% RSLogix 500 project DynamicDataExchange.RSS, saved by version 8.30.00.16 %
PROJECT "SIM_PLC"    % processor: Bul.1763 MicroLogix 1100 Series B %

PROGRAM FILES
  LAD 2 "MAIN"  2 rungs
  LAD 3 "CTRL LOGIC"  9 rungs

DATA FILES
  O0 OUTPUT  4 elements
  I1 INPUT  6 elements
  S2 STATUS  66 elements
  B3 BINARY  1 elements
  T4 TIMER  1 elements
  C5 COUNTER  5 elements
  R6 CONTROL  1 elements
  N7 INTEGER  4 elements
  F8 FLOAT  1 elements
  ST9 STRING  8 elements

LADDER 2 "MAIN"
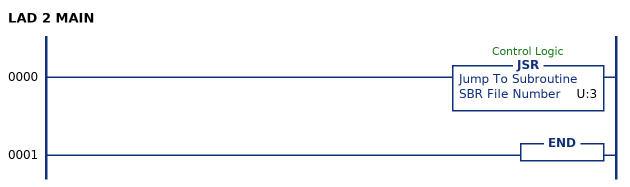
% Rung: 0 %
SOR JSR U:3 EOR
%   U:3  "Control Logic" %
% Rung: 1 %
SOR END EOR

LADDER 3 "CTRL LOGIC"
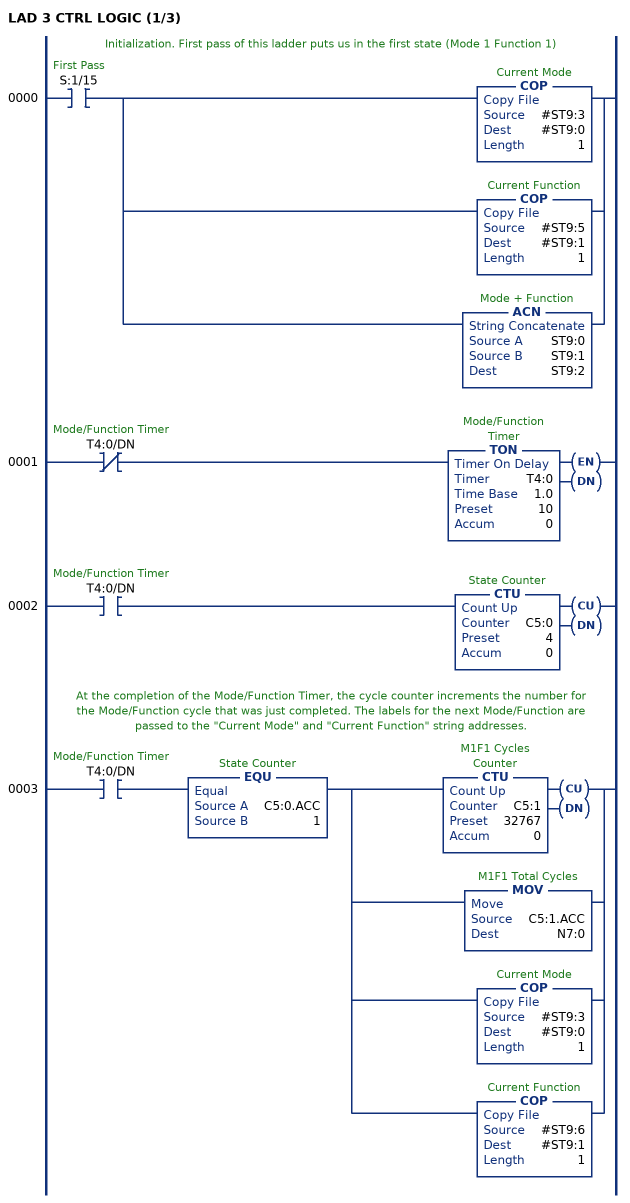
% Rung: 0 %
% Initialization. First pass of this ladder puts us in the first state (Mode 1 Function 1) %
SOR XIC S:1/15 BST COP #ST9:3 #ST9:0 1 NXB COP #ST9:5 #ST9:1 1 NXB ACN ST9:0 ST9:1 ST9:2 BND EOR
%   S:1/15  "First Pass" %
%   ST9:0  "Current Mode" %
%   ST9:1  "Current Function" %
%   ST9:2  "Mode + Function" %
% Rung: 1 %
SOR XIO T4:0/DN TON T4:0 1.0 10 0 EOR
%   T4:0  "Mode/Function Timer" %
% Rung: 2 %
SOR XIC T4:0/DN CTU C5:0 4 0 EOR
%   T4:0  "Mode/Function Timer" %
%   C5:0  "State Counter" %
% Rung: 3 %
% At the completion of the Mode/Function Timer, the cycle counter increments the number for the Mode/Function cycle that was just completed. The labels for the next Mode/Function are passed to the "Current Mode" and "Current Function" string addresses. %
SOR XIC T4:0/DN EQU C5:0.ACC 1 BST CTU C5:1 32767 0 NXB MOV C5:1.ACC N7:0 NXB COP #ST9:3 #ST9:0 1 NXB COP #ST9:6 #ST9:1 1 BND EOR
%   T4:0  "Mode/Function Timer" %
%   C5:0  "State Counter" %
%   C5:1  "M1F1 Cycles Counter" %
%   N7:0  "M1F1 Total Cycles" %
%   ST9:0  "Current Mode" %
%   ST9:1  "Current Function" %

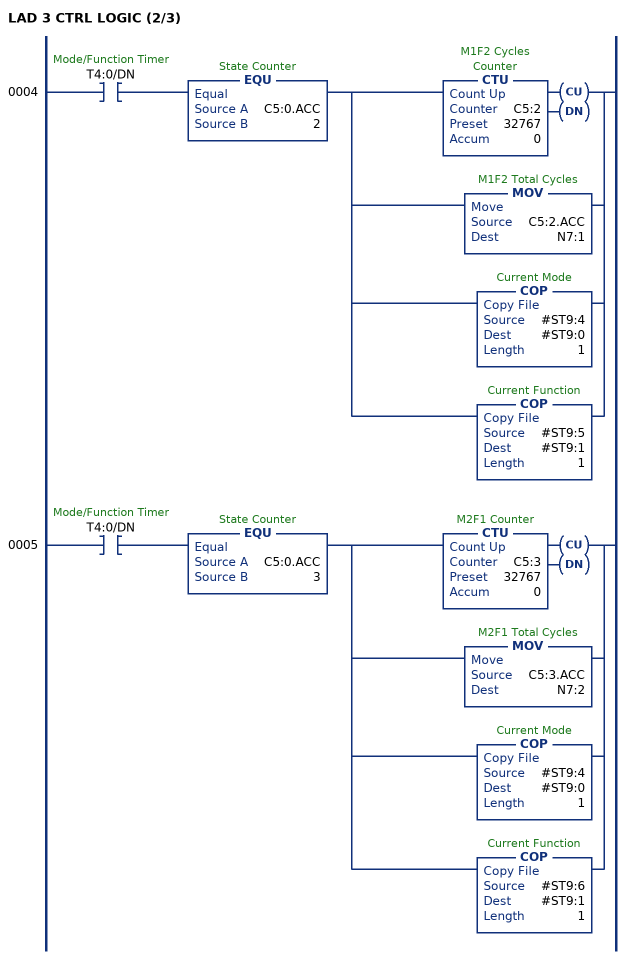
% Rung: 4 %
SOR XIC T4:0/DN EQU C5:0.ACC 2 BST CTU C5:2 32767 0 NXB MOV C5:2.ACC N7:1 NXB COP #ST9:4 #ST9:0 1 NXB COP #ST9:5 #ST9:1 1 BND EOR
%   T4:0  "Mode/Function Timer" %
%   C5:0  "State Counter" %
%   C5:2  "M1F2 Cycles Counter" %
%   N7:1  "M1F2 Total Cycles" %
%   ST9:0  "Current Mode" %
%   ST9:1  "Current Function" %
% Rung: 5 %
SOR XIC T4:0/DN EQU C5:0.ACC 3 BST CTU C5:3 32767 0 NXB MOV C5:3.ACC N7:2 NXB COP #ST9:4 #ST9:0 1 NXB COP #ST9:6 #ST9:1 1 BND EOR
%   T4:0  "Mode/Function Timer" %
%   C5:0  "State Counter" %
%   C5:3  "M2F1 Counter" %
%   N7:2  "M2F1 Total Cycles" %
%   ST9:0  "Current Mode" %
%   ST9:1  "Current Function" %

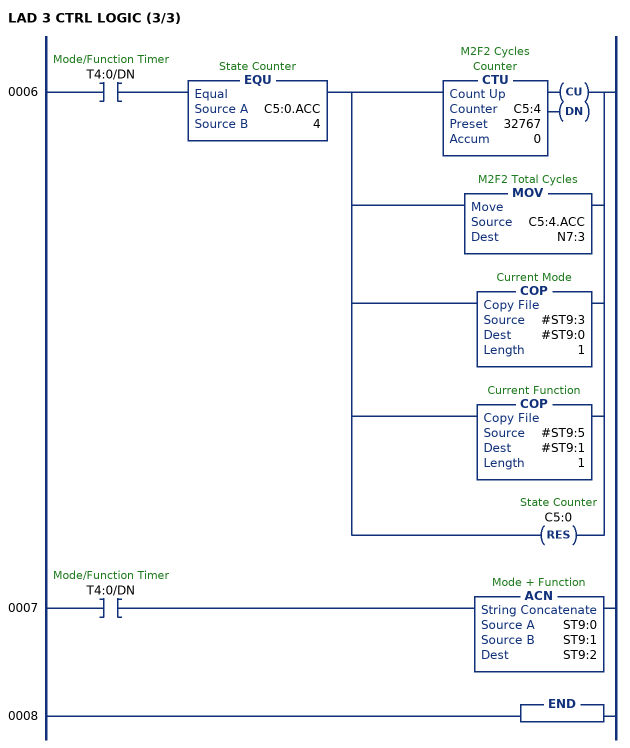
% Rung: 6 %
SOR XIC T4:0/DN EQU C5:0.ACC 4 BST CTU C5:4 32767 0 NXB MOV C5:4.ACC N7:3 NXB COP #ST9:3 #ST9:0 1 NXB COP #ST9:5 #ST9:1 1 NXB RES C5:0 BND EOR
%   T4:0  "Mode/Function Timer" %
%   C5:0  "State Counter" %
%   C5:4  "M2F2 Cycles Counter" %
%   N7:3  "M2F2 Total Cycles" %
%   ST9:0  "Current Mode" %
%   ST9:1  "Current Function" %
% Rung: 7 %
SOR XIC T4:0/DN ACN ST9:0 ST9:1 ST9:2 EOR
%   T4:0  "Mode/Function Timer" %
%   ST9:0  "Current Mode" %
%   ST9:1  "Current Function" %
%   ST9:2  "Mode + Function" %
% Rung: 8 %
SOR END EOR

DATA TABLE (non-zero values as saved)
DATA T4
% .PRE .ACC %
% T4:0 % 10 0
DATA C5
% .PRE .ACC %
% C5:0 % 4 0
% C5:1 % 32767 0
% C5:2 % 32767 0
% C5:3 % 32767 0
% C5:4 % 32767 0
DATA ST9
% ST9:3 % "M1"
% ST9:4 % "M2"
% ST9:5 % "F1"
% ST9:6 % "F2"
